FUNCTION_BLOCK FB_GCSpinAxisMoveAbsServiceTests EXTENDS TcUnit.FB_TestSuite

DelayedDoneCompletesAndReleasesAxis();
StopAndResetErrorsReachRecoverableAbortedState();

METHOD DelayedDoneCompletesAndReleasesAxis
VAR_INST
	FakeAxis : FB_FakeAxis_BaseUnit;
	Axis : I_Axis_BaseUnit;
	Service : FB_GCSpinAxisMoveAbsServices;
	Ctrl : ST_PML_Base_In;
	Param : ST_GCSpinAxisMoveAbsParam;
	CallRecord : ST_FakeAxisCall;
	nPhase : UINT;
END_VAR
TEST('DelayedDoneCompletesAndReleasesAxis');

CASE nPhase OF
	0:
		FakeAxis.M_ResetScenario();
		Axis := FakeAxis;
		Param.Position := 125.25;
		Param.Velocity := 15;
		Param.Acceleration := 25;
		Param.Deceleration := 35;
		AssertTrue(Condition := FakeAxis.M_QueueResult(Operation := E_FakeAxisOperation.MoveAbs, AfterActiveCycles := 2, Done := TRUE, InVelocity := FALSE, Error := FALSE, ErrorId := 0), Message := 'MoveAbs Done script must be accepted.');
		FakeAxis.M_CyclicUpdate();
		Service(PackMLIn := Ctrl, Param := Param, Axis_BaseUnit := Axis, ResourceOwnerId := 21);
		nPhase := 1;
	1:
		Ctrl.eCommand := E_PackMLCommand.Clear;
		Ctrl.bCommandChangeRequest := TRUE;
		FakeAxis.M_CyclicUpdate();
		Service(PackMLIn := Ctrl, Param := Param, Axis_BaseUnit := Axis, ResourceOwnerId := 21);
		Ctrl.bCommandChangeRequest := FALSE;
		FakeAxis.M_CyclicUpdate();
		Service(PackMLIn := Ctrl, Param := Param, Axis_BaseUnit := Axis, ResourceOwnerId := 21);
		Ctrl.eCommand := E_PackMLCommand.Reset;
		Ctrl.bCommandChangeRequest := TRUE;
		FakeAxis.M_CyclicUpdate();
		Service(PackMLIn := Ctrl, Param := Param, Axis_BaseUnit := Axis, ResourceOwnerId := 21);
		nPhase := 2;
	2:
		Ctrl.bCommandChangeRequest := FALSE;
		FakeAxis.M_CyclicUpdate();
		Service(PackMLIn := Ctrl, Param := Param, Axis_BaseUnit := Axis, ResourceOwnerId := 21);
		Ctrl.eCommand := E_PackMLCommand.Start;
		Ctrl.bCommandChangeRequest := TRUE;
		FakeAxis.M_CyclicUpdate();
		Service(PackMLIn := Ctrl, Param := Param, Axis_BaseUnit := Axis, ResourceOwnerId := 21);
		Ctrl.bCommandChangeRequest := FALSE;
		AssertTrue(Condition := Service.PackMLOut.eStateCurrent = E_PackMLState.Execute, Message := 'Valid MoveAbs must enter Execute.');
		nPhase := 3;
	3:
		FakeAxis.M_CyclicUpdate();
		Service(PackMLIn := Ctrl, Param := Param, Axis_BaseUnit := Axis, ResourceOwnerId := 21);
		AssertTrue(Condition := FakeAxis.M_GetCall(Index := FakeAxis.HistoryCount, CallRecord => CallRecord), Message := 'MoveAbs command must be recorded.');
		AssertTrue(Condition := CallRecord.Execute, Message := 'MoveAbs must assert Execute.');
		AssertTrue(Condition := (CallRecord.Position = 125.25) AND (CallRecord.Velocity = 15), Message := 'MoveAbs position and velocity must be preserved.');
		nPhase := 4;
	4:
		FakeAxis.M_CyclicUpdate();
		Service(PackMLIn := Ctrl, Param := Param, Axis_BaseUnit := Axis, ResourceOwnerId := 21);
		AssertTrue(Condition := Axis.M_IsResourceOwner(OwnerId := 21), Message := 'MoveAbs must retain ownership while Done is pending.');
		nPhase := 5;
	5:
		FakeAxis.M_CyclicUpdate();
		Service(PackMLIn := Ctrl, Param := Param, Axis_BaseUnit := Axis, ResourceOwnerId := 21);
		AssertTrue(Condition := Service.PackMLOut.eStateCurrent = E_PackMLState.Completing, Message := 'Delayed Done must enter Completing.');
		nPhase := 6;
	6:
		FakeAxis.M_CyclicUpdate();
		Service(PackMLIn := Ctrl, Param := Param, Axis_BaseUnit := Axis, ResourceOwnerId := 21);
		AssertTrue(Condition := Service.PackMLOut.eStateCurrent = E_PackMLState.Complete, Message := 'Completing must finish at Complete.');
		AssertFalse(Condition := Axis.M_IsResourceOwner(OwnerId := 21), Message := 'Complete must release Axis ownership.');
		AssertTrue(Condition := FakeAxis.M_GetCall(Index := FakeAxis.HistoryCount, CallRecord => CallRecord), Message := 'MoveAbs withdrawal must be recorded.');
		AssertFalse(Condition := CallRecord.Execute, Message := 'Completing must withdraw MoveAbs Execute.');
		nPhase := 0;
		TEST_FINISHED();
END_CASE
END_METHOD

METHOD StopAndResetErrorsReachRecoverableAbortedState
VAR_INST
	FakeAxis : FB_FakeAxis_BaseUnit;
	Axis : I_Axis_BaseUnit;
	Service : FB_GCSpinAxisMoveAbsServices;
	Ctrl : ST_PML_Base_In;
	Param : ST_GCSpinAxisMoveAbsParam;
	nPhase : UINT;
END_VAR
TEST('StopAndResetErrorsReachRecoverableAbortedState');

CASE nPhase OF
	0:
		FakeAxis.M_ResetScenario();
		Axis := FakeAxis;
		Param.Position := 50;
		Param.Velocity := 10;
		Param.Acceleration := 20;
		Param.Deceleration := 30;
		AssertTrue(Condition := FakeAxis.M_QueueResult(Operation := E_FakeAxisOperation.MoveAbs, AfterActiveCycles := 1, Done := FALSE, InVelocity := FALSE, Error := TRUE, ErrorId := 1), Message := 'MoveAbs Error must be queued.');
		AssertTrue(Condition := FakeAxis.M_QueueResult(Operation := E_FakeAxisOperation.Stop, AfterActiveCycles := 1, Done := FALSE, InVelocity := FALSE, Error := TRUE, ErrorId := 2), Message := 'Stop Error must be queued.');
		AssertTrue(Condition := FakeAxis.M_QueueResult(Operation := E_FakeAxisOperation.Reset, AfterActiveCycles := 1, Done := FALSE, InVelocity := FALSE, Error := TRUE, ErrorId := 3), Message := 'Reset Error must be queued.');
		FakeAxis.M_CyclicUpdate();
		Service(PackMLIn := Ctrl, Param := Param, Axis_BaseUnit := Axis, ResourceOwnerId := 22);
		nPhase := 1;
	1:
		Ctrl.eCommand := E_PackMLCommand.Clear;
		Ctrl.bCommandChangeRequest := TRUE;
		FakeAxis.M_CyclicUpdate();
		Service(PackMLIn := Ctrl, Param := Param, Axis_BaseUnit := Axis, ResourceOwnerId := 22);
		Ctrl.bCommandChangeRequest := FALSE;
		FakeAxis.M_CyclicUpdate();
		Service(PackMLIn := Ctrl, Param := Param, Axis_BaseUnit := Axis, ResourceOwnerId := 22);
		Ctrl.eCommand := E_PackMLCommand.Reset;
		Ctrl.bCommandChangeRequest := TRUE;
		FakeAxis.M_CyclicUpdate();
		Service(PackMLIn := Ctrl, Param := Param, Axis_BaseUnit := Axis, ResourceOwnerId := 22);
		nPhase := 2;
	2:
		Ctrl.bCommandChangeRequest := FALSE;
		FakeAxis.M_CyclicUpdate();
		Service(PackMLIn := Ctrl, Param := Param, Axis_BaseUnit := Axis, ResourceOwnerId := 22);
		Ctrl.eCommand := E_PackMLCommand.Start;
		Ctrl.bCommandChangeRequest := TRUE;
		FakeAxis.M_CyclicUpdate();
		Service(PackMLIn := Ctrl, Param := Param, Axis_BaseUnit := Axis, ResourceOwnerId := 22);
		Ctrl.bCommandChangeRequest := FALSE;
		FakeAxis.M_CyclicUpdate();
		Service(PackMLIn := Ctrl, Param := Param, Axis_BaseUnit := Axis, ResourceOwnerId := 22);
		nPhase := 3;
	3:
		FakeAxis.M_CyclicUpdate();
		Service(PackMLIn := Ctrl, Param := Param, Axis_BaseUnit := Axis, ResourceOwnerId := 22);
		AssertTrue(Condition := Service.Status.ServiceErrorId = E_GCSpinAxisMoveAbsErrorCode.MoveAbs_Error_During_Execute, Message := 'MoveAbs Error must request Stop.');
		nPhase := 4;
	4:
		FakeAxis.M_CyclicUpdate();
		Service(PackMLIn := Ctrl, Param := Param, Axis_BaseUnit := Axis, ResourceOwnerId := 22);
		AssertTrue(Condition := Axis.M_IsResourceOwner(OwnerId := 22), Message := 'Stop Pending/Error handling must retain ownership until Abort cleanup.');
		nPhase := 5;
	5:
		FakeAxis.M_CyclicUpdate();
		Service(PackMLIn := Ctrl, Param := Param, Axis_BaseUnit := Axis, ResourceOwnerId := 22);
		nPhase := 6;
	6:
		FakeAxis.M_CyclicUpdate();
		Service(PackMLIn := Ctrl, Param := Param, Axis_BaseUnit := Axis, ResourceOwnerId := 22);
		nPhase := 7;
	7:
		FakeAxis.M_CyclicUpdate();
		Service(PackMLIn := Ctrl, Param := Param, Axis_BaseUnit := Axis, ResourceOwnerId := 22);
		AssertTrue(Condition := Service.PackMLOut.eStateCurrent = E_PackMLState.Aborted, Message := 'Reset Error must terminate Aborting at Aborted.');
		AssertTrue(Condition := Service.Status.Error, Message := 'Reset Error must remain reported.');
		AssertTrue(Condition := Service.Status.ServiceErrorId = E_GCSpinAxisMoveAbsErrorCode.Error_While_Reset_Axis, Message := 'Reset Error must use the new error code.');
		AssertFalse(Condition := Axis.M_IsResourceOwner(OwnerId := 22), Message := 'Reset Error must release ownership.');
		nPhase := 0;
		TEST_FINISHED();
END_CASE
END_METHOD

END_FUNCTION_BLOCK

(* stored: Version 1.1.0.1, ProductVersion 3.1.4026.18
   POU FB_GCSpinAxisMoveAbsServiceTests: Id {976b21c2-7581-4c58-b755-8768083df5a7}, SpecialFunc None
   Method DelayedDoneCompletesAndReleasesAxis: Id {7f47f8ae-15f2-4e92-b2c7-8cd52301a876}
   Method StopAndResetErrorsReachRecoverableAbortedState: Id {b9229082-c8d5-4882-95e8-07156341bc38} *)
